{attribute 'linkalways'}
{attribute 'no_explicit_call' := 'do not call this POU directly'}
FUNCTION_BLOCK CyclicCallback IMPLEMENTS I_Callback
VAR
	target : I_CyclicCalled;
END_VAR

METHOD FB_init : BOOL
VAR_INPUT
	bInitRetains : BOOL; // if TRUE, the retain variables are initialized (warm start / cold start)
	bInCopyCode : BOOL;  // if TRUE, the instance afterwards gets moved into the copy code (online change)
	Target : I_CyclicCalled;
END_VAR
this^.target := Target;
END_METHOD

METHOD PUBLIC Update
VAR_INPUT
	Event : I_Event;
END_VAR
IF target <> 0 THEN
	target.CyclicCall();
END_IF
END_METHOD

END_FUNCTION_BLOCK

(* stored: Version 1.1.0.1, ProductVersion 3.1.4024.11
   POU CyclicCallback: Id {9f56da02-9969-4a62-b3ab-89de78f9213e}, SpecialFunc None
   Folder Constructor: Id {233d67cf-f5ec-42c2-8221-8a5683f18ef1}
   Method FB_init: Id {ab963e7e-1c1f-4632-a9d5-57230918bf9f}
   Method Update: Id {b0c3b4d3-42f6-4a0a-b433-de659224cd84} *)
